// TIA Portal project "FactoryIO_Template_S7-1200_V16_V16" (V16)
// Vorlageprojekt für das Buch mit Zielsystem S7-1200

(* hardware
DEVICE "S7-1200-Station_1"  S7-1200 Station
   slot 0: "Baugruppenträger_0"  Rack  V1.0
   slot 1: "PLC_1"  CPU 1211C DC/DC/DC  6ES7 211-1AE40-0XB0  V4.1
*)

// ===== PLC "PLC_1"  CPU 1211C DC/DC/DC =====

VAR_GLOBAL   // PLC tag table "Standard-Variablentabelle"
   "start" AT %I0.0 : Bool;
   "stop" AT %I0.1 : Bool;
   "blue_sensor" AT %I0.2 : Bool;
   "Green_sensor" AT %I0.3 : Bool;
   "Diff_1_BR" AT %I0.4 : Bool;
   "Diff_2_BR" AT %I0.5 : Bool;
   "Diff_3_BL" AT %I0.6 : Bool;
   "Diff_4_BL" AT %I0.7 : Bool;
   "Diff_5_AR" AT %I1.0 : Bool;
   "Diff_6_AL" AT %I1.1 : Bool;
   "Grap_detector_1" AT %I1.4 : Bool;
   "Grap_detector_2" AT %I1.5 : Bool;
   "Belt_main_C" AT %Q0.0 : Bool;
   "Belt_Box_Right" AT %Q0.1 : Bool;
   "Belt_Box_left" AT %Q0.2 : Bool;
   "Belt_Right_GRE" AT %Q0.3 : Bool;
   "Belt_Left_RED" AT %Q0.4 : Bool;
   "Selector_on" AT %Q0.5 : Bool;
   "Selector_Left" AT %Q0.7 : Bool;
   "Selector_Right" AT %Q0.6 : Bool;
   "Move_V_1" AT %Q1.0 : Bool;
   "Move_V_2" AT %Q1.1 : Bool;
   "Grap_1" AT %Q1.2 : Bool;
   "Grap_2" AT %Q1.3 : Bool;
   "Move_H_1" AT %Q1.4 : Bool;
   "Move_H_2" AT %Q1.5 : Bool;
   "X" AT %M0.0 : Bool;
   "reach_target_1_H" AT %I1.6 : Bool;
   "reach_target_2_H" AT %I1.7 : Bool;
   "reach_target_1_V" AT %I1.2 : Bool;
   "reach_target_2_V" AT %I1.3 : Bool;
   "stop_grep_1" AT %M0.3 : Bool;
   "stop_grep_2" AT %M0.4 : Bool;
   "Tag_1" AT %M0.5 : Bool;
   "Tag_2" AT %M0.6 : Bool;
   "Tag_3" AT %M0.7 : Bool;
   "ungrep_2" AT %M1.0 : Bool;
   "ungrep_1" AT %M1.1 : Bool;
   "Tag_4" AT %M1.5 : Bool;
   "Tag_5" AT %M1.6 : Bool;
   "Tag_6" AT %M1.3 : Bool;
   "Tag_7" AT %M1.7 : Bool;
END_VAR

// folder: System blocks/Program resources

DATA_BLOCK "T"   // DB1
{ S7_Optimized_Access := 'TRUE' }
AUTHOR : Simatic
FAMILY : IEC
NAME : IEC_TMR
VERSION : 1.0
// stored: InstanceOfName IEC_TIMER
"IEC_TIMER"
BEGIN
END_DATA_BLOCK

DATA_BLOCK "t_off"   // DB2
{ S7_Optimized_Access := 'TRUE' }
AUTHOR : Simatic
FAMILY : IEC
NAME : IEC_TMR
VERSION : 1.0
// stored: InstanceOfName IEC_TIMER
"IEC_TIMER"
BEGIN
END_DATA_BLOCK

DATA_BLOCK "t_off_2"   // DB3
{ S7_Optimized_Access := 'TRUE' }
AUTHOR : Simatic
FAMILY : IEC
NAME : IEC_TMR
VERSION : 1.0
// stored: InstanceOfName IEC_TIMER
"IEC_TIMER"
BEGIN
END_DATA_BLOCK

// folder: (top level)

FUNCTION "MHJ-PLC-Lab-Function-S71200" : Void   // FC9000, SCL
{ S7_Optimized_Access := 'TRUE' }
VERSION : 0.1
   VAR_TEMP
      rdTimeReturn : Int;
      outputTime : DTL;
      SyncVal : Byte;
      forVal : Int;
      forVal_2 : Int;
      Value : Byte;
   END_VAR
   VAR CONSTANT
      CompVal : Byte := 16#34;
      Value_01 : Byte := 16#11;
      Value_01_DW : DWord := 16#A165_D992;
      Value_02_DW : DWord := 16#58BE_4401;
   END_VAR
BEGIN

   #Value:=PEEK(area := 16#82,
        dbNumber := 0,
        byteOffset := 511);
   #Value := #Value + 1;

   POKE(area := 16#82,
        dbNumber := 0,
        byteOffset := 511,
        value := #Value);

   POKE(area:=16#81,
        dbNumber:=0,
        byteOffset:=1016,
        value:=#Value_01_DW);
   POKE(area := 16#81,
        dbNumber := 0,
        byteOffset := 1020,
        value := #Value_02_DW);

   POKE(area := 16#81,
        dbNumber := 0,
        byteOffset := 511,
        value := B#16#00);

   FOR #forVal := 0 TO 120 DO
       FOR #forVal_2:=0 TO 10 DO
           #rdTimeReturn:=RD_SYS_T(#outputTime);
           #rdTimeReturn := WR_SYS_T(#outputTime);
           #rdTimeReturn := RD_SYS_T(#outputTime);
           #rdTimeReturn := WR_SYS_T(#outputTime);
       END_FOR;
       #SyncVal:= PEEK(area := 16#81,
                      dbNumber := 0,
                      byteOffset := 511);
       IF #SyncVal = #CompVal THEN
          GOTO M_1;
       END_IF;
   END_FOR;
   RETURN;

   M_1:
   POKE(area := 16#81,
        dbNumber := 0,
        byteOffset := 511,
        value := B#16#0);
END_FUNCTION

ORGANIZATION_BLOCK "Main"   // OB1, LAD, ProgramCycle
TITLE = "Main Program Sweep (Cycle)"
{ S7_Optimized_Access := 'TRUE' }
VERSION : 0.1
   VAR_INPUT
      Initial_Call : Bool;   // Initial call of this OB
      Remanence : Bool;   // =True, if remanent data are available
   END_VAR
   VAR_TEMP   // added for the SCL form of the ladder/FBD networks
      _w1 : Bool;
   END_VAR
BEGIN

REGION Network 1: Konnektierungsbaustein für PLC-Lab
   // Im Netzwerk 1 wird der Konnektierungsbaustein für PLC-Lab aufgerufen.
   // Dieser Aufruf darf nicht entfernt werden!
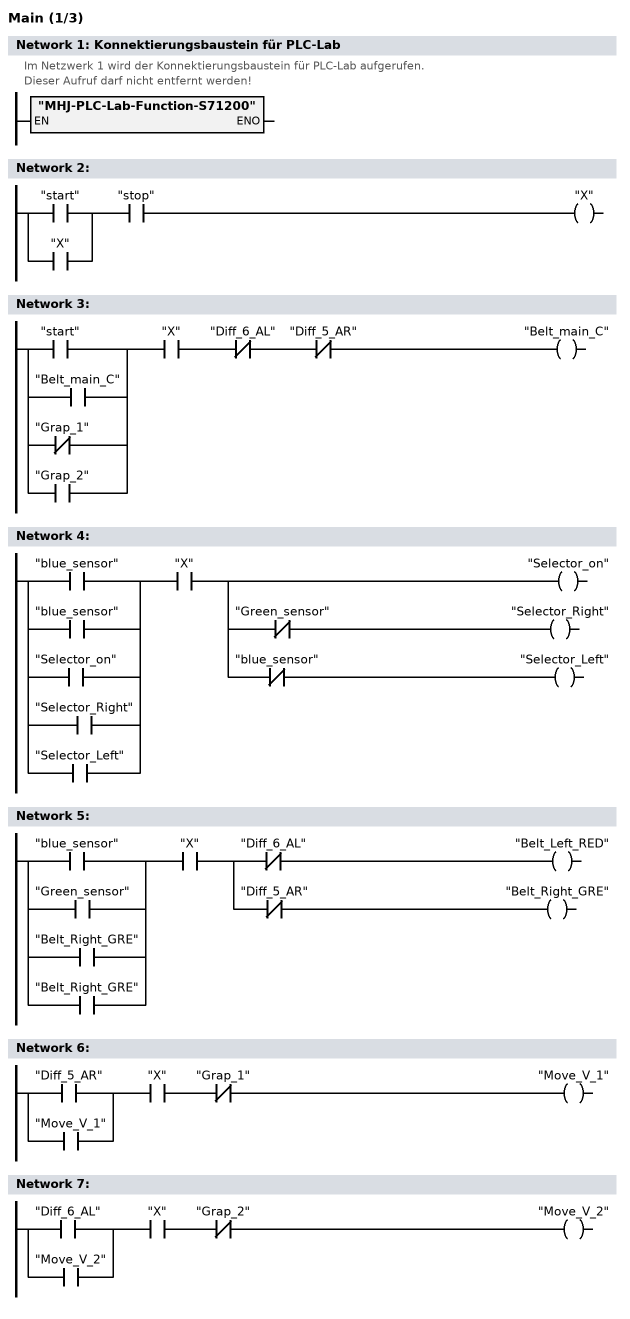
   RUNG wire#powerrail
      "MHJ-PLC-Lab-Function-S71200"()
   END_RUNG
   // the same network as SCL:
   "MHJ-PLC-Lab-Function-S71200"();
END_REGION

REGION Network 2
   RUNG wire#powerrail
      Contact( "start" )
      wire#w1
      Contact( "stop" )
      Coil( "X" )
   END_RUNG
   RUNG wire#powerrail
      Contact( "X" )
   END_RUNG wire#w1
   // the same network as SCL:
   "X" := ("start" OR "X") AND "stop";
END_REGION

REGION Network 3
   RUNG wire#powerrail
      Contact( "start" )
      wire#w1
      Contact( "X" )
      I_Contact( "Diff_6_AL" )
      I_Contact( "Diff_5_AR" )
      Coil( "Belt_main_C" )
   END_RUNG
   RUNG wire#powerrail
      Contact( "Belt_main_C" )
   END_RUNG wire#w1
   RUNG wire#powerrail
      I_Contact( "Grap_1" )
   END_RUNG wire#w1
   RUNG wire#powerrail
      Contact( "Grap_2" )
   END_RUNG wire#w1
   // the same network as SCL:
   "Belt_main_C" := ("start" OR "Belt_main_C" OR NOT "Grap_1" OR "Grap_2") AND "X" AND NOT "Diff_6_AL" AND NOT "Diff_5_AR";
END_REGION

REGION Network 4
   RUNG wire#powerrail
      Contact( "blue_sensor" )
      wire#w1
      Contact( "X" )
      wire#w2
      Coil( "Selector_on" )
   END_RUNG
   RUNG wire#powerrail
      Contact( "blue_sensor" )
   END_RUNG wire#w1
   RUNG wire#powerrail
      Contact( "Selector_on" )
   END_RUNG wire#w1
   RUNG wire#powerrail
      Contact( "Selector_Right" )
   END_RUNG wire#w1
   RUNG wire#powerrail
      Contact( "Selector_Left" )
   END_RUNG wire#w1
   RUNG wire#w2
      I_Contact( "Green_sensor" )
      Coil( "Selector_Right" )
   END_RUNG
   RUNG wire#w2
      I_Contact( "blue_sensor" )
      Coil( "Selector_Left" )
   END_RUNG
   // the same network as SCL:
   "Selector_on" := ("blue_sensor" OR "blue_sensor" OR "Selector_on" OR "Selector_Right" OR "Selector_Left") AND "X";
   "Selector_Right" := "Selector_on" AND NOT "Green_sensor";
   "Selector_Left" := "Selector_on" AND NOT "blue_sensor";
END_REGION

REGION Network 5
   RUNG wire#powerrail
      Contact( "blue_sensor" )
      wire#w1
      Contact( "X" )
      wire#w2
      I_Contact( "Diff_6_AL" )
      Coil( "Belt_Left_RED" )
   END_RUNG
   RUNG wire#powerrail
      Contact( "Green_sensor" )
   END_RUNG wire#w1
   RUNG wire#powerrail
      Contact( "Belt_Right_GRE" )
   END_RUNG wire#w1
   RUNG wire#powerrail
      Contact( "Belt_Right_GRE" )
   END_RUNG wire#w1
   RUNG wire#w2
      I_Contact( "Diff_5_AR" )
      Coil( "Belt_Right_GRE" )
   END_RUNG
   // the same network as SCL:
   #_w1 := ("blue_sensor" OR "Green_sensor" OR "Belt_Right_GRE" OR "Belt_Right_GRE") AND "X";
   "Belt_Left_RED" := #_w1 AND NOT "Diff_6_AL";
   "Belt_Right_GRE" := #_w1 AND NOT "Diff_5_AR";
END_REGION

REGION Network 6
   RUNG wire#powerrail
      Contact( "Diff_5_AR" )
      wire#w1
      Contact( "X" )
      I_Contact( "Grap_1" )
      Coil( "Move_V_1" )
   END_RUNG
   RUNG wire#powerrail
      Contact( "Move_V_1" )
   END_RUNG wire#w1
   // the same network as SCL:
   "Move_V_1" := ("Diff_5_AR" OR "Move_V_1") AND "X" AND NOT "Grap_1";
END_REGION

REGION Network 7
   RUNG wire#powerrail
      Contact( "Diff_6_AL" )
      wire#w1
      Contact( "X" )
      I_Contact( "Grap_2" )
      Coil( "Move_V_2" )
   END_RUNG
   RUNG wire#powerrail
      Contact( "Move_V_2" )
   END_RUNG wire#w1
   // the same network as SCL:
   "Move_V_2" := ("Diff_6_AL" OR "Move_V_2") AND "X" AND NOT "Grap_2";
END_REGION

REGION Network 8
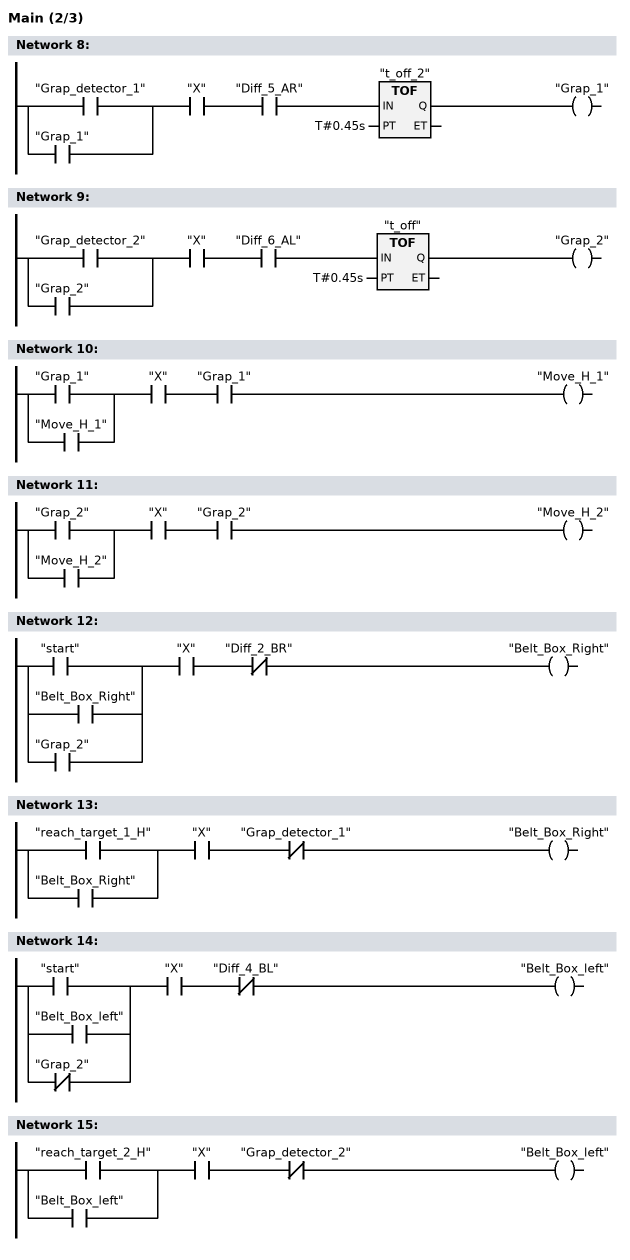
   "t_off_2".TOF(IN := ("Grap_detector_1" OR "Grap_1") AND "X" AND "Diff_5_AR", PT := T#0.45s);
   "Grap_1" := "t_off_2".Q;
END_REGION

REGION Network 9
   "t_off".TOF(IN := ("Grap_detector_2" OR "Grap_2") AND "X" AND "Diff_6_AL", PT := T#0.45s);
   "Grap_2" := "t_off".Q;
END_REGION

REGION Network 10
   RUNG wire#powerrail
      Contact( "Grap_1" )
      wire#w1
      Contact( "X" )
      Contact( "Grap_1" )
      Coil( "Move_H_1" )
   END_RUNG
   RUNG wire#powerrail
      Contact( "Move_H_1" )
   END_RUNG wire#w1
   // the same network as SCL:
   "Move_H_1" := ("Grap_1" OR "Move_H_1") AND "X" AND "Grap_1";
END_REGION

REGION Network 11
   RUNG wire#powerrail
      Contact( "Grap_2" )
      wire#w1
      Contact( "X" )
      Contact( "Grap_2" )
      Coil( "Move_H_2" )
   END_RUNG
   RUNG wire#powerrail
      Contact( "Move_H_2" )
   END_RUNG wire#w1
   // the same network as SCL:
   "Move_H_2" := ("Grap_2" OR "Move_H_2") AND "X" AND "Grap_2";
END_REGION

REGION Network 12
   RUNG wire#powerrail
      Contact( "start" )
      wire#w1
      Contact( "X" )
      I_Contact( "Diff_2_BR" )
      Coil( "Belt_Box_Right" )
   END_RUNG
   RUNG wire#powerrail
      Contact( "Belt_Box_Right" )
   END_RUNG wire#w1
   RUNG wire#powerrail
      Contact( "Grap_2" )
   END_RUNG wire#w1
   // the same network as SCL:
   "Belt_Box_Right" := ("start" OR "Belt_Box_Right" OR "Grap_2") AND "X" AND NOT "Diff_2_BR";
END_REGION

REGION Network 13
   RUNG wire#powerrail
      Contact( "reach_target_1_H" )
      wire#w1
      Contact( "X" )
      I_Contact( "Grap_detector_1" )
      Coil( "Belt_Box_Right" )
   END_RUNG
   RUNG wire#powerrail
      Contact( "Belt_Box_Right" )
   END_RUNG wire#w1
   // the same network as SCL:
   "Belt_Box_Right" := ("reach_target_1_H" OR "Belt_Box_Right") AND "X" AND NOT "Grap_detector_1";
END_REGION

REGION Network 14
   RUNG wire#powerrail
      Contact( "start" )
      wire#w1
      Contact( "X" )
      I_Contact( "Diff_4_BL" )
      Coil( "Belt_Box_left" )
   END_RUNG
   RUNG wire#powerrail
      Contact( "Belt_Box_left" )
   END_RUNG wire#w1
   RUNG wire#powerrail
      I_Contact( "Grap_2" )
   END_RUNG wire#w1
   // the same network as SCL:
   "Belt_Box_left" := ("start" OR "Belt_Box_left" OR NOT "Grap_2") AND "X" AND NOT "Diff_4_BL";
END_REGION

REGION Network 15
   RUNG wire#powerrail
      Contact( "reach_target_2_H" )
      wire#w1
      Contact( "X" )
      I_Contact( "Grap_detector_2" )
      Coil( "Belt_Box_left" )
   END_RUNG
   RUNG wire#powerrail
      Contact( "Belt_Box_left" )
   END_RUNG wire#w1
   // the same network as SCL:
   "Belt_Box_left" := ("reach_target_2_H" OR "Belt_Box_left") AND "X" AND NOT "Grap_detector_2";
END_REGION

REGION Network 16
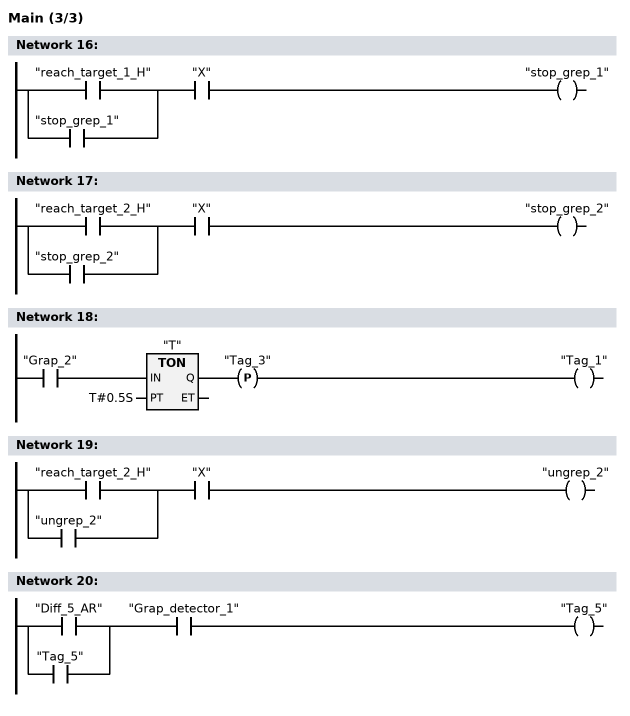
   RUNG wire#powerrail
      Contact( "reach_target_1_H" )
      wire#w1
      Contact( "X" )
      Coil( "stop_grep_1" )
   END_RUNG
   RUNG wire#powerrail
      Contact( "stop_grep_1" )
   END_RUNG wire#w1
   // the same network as SCL:
   "stop_grep_1" := ("reach_target_1_H" OR "stop_grep_1") AND "X";
END_REGION

REGION Network 17
   RUNG wire#powerrail
      Contact( "reach_target_2_H" )
      wire#w1
      Contact( "X" )
      Coil( "stop_grep_2" )
   END_RUNG
   RUNG wire#powerrail
      Contact( "stop_grep_2" )
   END_RUNG wire#w1
   // the same network as SCL:
   "stop_grep_2" := ("reach_target_2_H" OR "stop_grep_2") AND "X";
END_REGION

REGION Network 18
   "T".TON(IN := "Grap_2", PT := T#0.5S);
   #_w1 := "T".Q AND NOT "Tag_3";   // rising edge
   "Tag_3" := "T".Q;
   "Tag_1" := #_w1;
END_REGION

REGION Network 19
   RUNG wire#powerrail
      Contact( "reach_target_2_H" )
      wire#w1
      Contact( "X" )
      Coil( "ungrep_2" )
   END_RUNG
   RUNG wire#powerrail
      Contact( "ungrep_2" )
   END_RUNG wire#w1
   // the same network as SCL:
   "ungrep_2" := ("reach_target_2_H" OR "ungrep_2") AND "X";
END_REGION

REGION Network 20
   RUNG wire#powerrail
      Contact( "Diff_5_AR" )
      wire#w1
      Contact( "Grap_detector_1" )
      Coil( "Tag_5" )
   END_RUNG
   RUNG wire#powerrail
      Contact( "Tag_5" )
   END_RUNG wire#w1
   // the same network as SCL:
   "Tag_5" := ("Diff_5_AR" OR "Tag_5") AND "Grap_detector_1";
END_REGION
END_ORGANIZATION_BLOCK